FUNCTION WRITE_PROTECTED_USINT
VAR_INPUT
    Ptr : POINTER TO USINT;
    Value : USINT;
END_VAR

Ptr^ := Value;

END_FUNCTION

(* stored: Version 1.1.0.1, ProductVersion 3.1.4024.9
   POU WRITE_PROTECTED_USINT: Id {f1079ab8-dc5a-06e1-34a2-495bc4f858b4}, SpecialFunc None *)
